          sync()
        end
        $ 4413 "Set CO[1]=Apagar"
        set_configurable_digital_out(1, False)
        $ 4414 "subir" "breakAfter"
        movel(subir, a=0.015, v=0.015)
        $ 4415 "bajada_broca≔pose_sub(bajada_broca, bajada)"
        global bajada_broca= pose_sub (bajada_broca, bajada)
        Loop_88 = Loop_88 + 1
      end
      $ 4416 "Direction: Base Z+"
      global move_thread_flag_4416=0
      thread move_thread_4416():
        enter_critical
        move_thread_flag_4416 = 1
        local towardsPos=calculate_point_to_move_towards(p[0.0,0.0,0.0,0.0,0.0,0.0], [0.0,0.0,1.0], 0.08)
        movel(towardsPos, a=0.15, v=0.1)
        move_thread_flag_4416 = 2
        exit_critical
      end
      move_thread_flag_4416 = 0
      move_thread_han_4416 = run move_thread_4416()
      while (True):
        sleep(1.0E-10)
        if (move_thread_flag_4416 > 1):
          join move_thread_han_4416
          $ 4417 "Until (distance)"
          break
        end
        sync()
      end
      $ 4418 "Set CO[1]=Apagar"
      set_configurable_digital_out(1, False)
      $ 4419 "barreno_actual≔barreno_actual+1"
      global barreno_actual=barreno_actual+1
    end
    $ 4422 "Popup: Linea23 con chica Terminada!"
    popup("Linea23 con chica Terminada!", "Mensaje", False, False, blocking=True)
    $ 4423 "Linea24"
    $ 4424 "Marcar_puntos"
    $ 4425 "MoveL"
    $ 4426 "Linea24_A" "breakAfter"
    movel(Linea24_A_p, a=0.5, v=0.1)
    $ 4427 "bajada_comprobacion"
    $ 4428 "Direction: Base Z-"
    global move_thread_flag_4428=0
    thread move_thread_4428():
      enter_critical
      move_thread_flag_4428 = 1
      local towardsPos=calculate_point_to_move_towards(p[0.0,0.0,0.0,0.0,0.0,0.0], [0.0,0.0,-1.0], 0.071)
      movel(towardsPos, a=0.15, v=0.1)
      move_thread_flag_4428 = 2
      exit_critical
    end
    move_thread_flag_4428 = 0
    move_thread_han_4428 = run move_thread_4428()
    while (True):
      sleep(1.0E-10)
      if (move_thread_flag_4428 > 1):
        join move_thread_han_4428
        $ 4429 "Until (distance)"
        break
      end
      sync()
    end
    $ 4430 "Direction: Base Z-"
    global move_thread_flag_4430=0
    thread move_thread_4430():
      enter_critical
      move_thread_flag_4430 = 1
      local towardsPos=calculate_point_to_move_towards(p[0.0,0.0,0.0,0.0,0.0,0.0], [0.0,0.0,-1.0], 1000.0)
      movel(towardsPos, a=0.007, v=0.007)
      move_thread_flag_4430 = 2
      exit_critical
    end
    move_thread_flag_4430 = 0
    move_thread_han_4430 = run move_thread_4430()
    while (True):
      local targetTcpDirection=get_target_tcp_speed()
      local stepsToRetract=tool_contact(direction=targetTcpDirection)
      if (stepsToRetract > 0):
        kill move_thread_han_4430
        stopl(0.02)
        local backTrackMovement=get_actual_joint_positions_history(stepsToRetract)
        local contactPose=get_forward_kin(backTrackMovement)
        local posDir=[targetTcpDirection[0],targetTcpDirection[1],targetTcpDirection[2]]
        local retractTo=contactPose
        if (norm(posDir) > 1e-6):
          local normalizedPosDir=normalize(posDir)
          local additionalRetraction=p[normalizedPosDir[0] * 0.0, normalizedPosDir[1] * 0.0, normalizedPosDir[2] * 0.0, 0, 0, 0]
          retractTo = pose_sub(contactPose, additionalRetraction)
        end
        movel(retractTo, a=0.02, v=0.1)
        $ 4431 "Until (tool_contact_detection)"
        break
      end
      sync()
    end
    $ 4432 "Direction: Base Z+"
    global move_thread_flag_4432=0
    thread move_thread_4432():
      enter_critical
      move_thread_flag_4432 = 1
      local towardsPos=calculate_point_to_move_towards(p[0.0,0.0,0.0,0.0,0.0,0.0], [0.0,0.0,1.0], 0.08)
      movel(towardsPos, a=0.15, v=0.1)
      move_thread_flag_4432 = 2
      exit_critical
    end
    move_thread_flag_4432 = 0
    move_thread_han_4432 = run move_thread_4432()
    while (True):
      sleep(1.0E-10)
      if (move_thread_flag_4432 > 1):
        join move_thread_han_4432
        $ 4433 "Until (distance)"
        break
      end
      sync()
    end
    $ 4434 "Linea24_B" "breakAfter"
    movel(Linea24_B_p, a=0.5, v=0.1)
    $ 4435 "bajada_comprobacion"
    $ 4436 "Direction: Base Z-"
    global move_thread_flag_4436=0
    thread move_thread_4436():
      enter_critical
      move_thread_flag_4436 = 1
      local towardsPos=calculate_point_to_move_towards(p[0.0,0.0,0.0,0.0,0.0,0.0], [0.0,0.0,-1.0], 0.071)
      movel(towardsPos, a=0.15, v=0.1)
      move_thread_flag_4436 = 2
      exit_critical
    end
    move_thread_flag_4436 = 0
    move_thread_han_4436 = run move_thread_4436()
    while (True):
      sleep(1.0E-10)
      if (move_thread_flag_4436 > 1):
        join move_thread_han_4436
        $ 4437 "Until (distance)"
        break
      end
      sync()
    end
    $ 4438 "Direction: Base Z-"
    global move_thread_flag_4438=0
    thread move_thread_4438():
      enter_critical
      move_thread_flag_4438 = 1
      local towardsPos=calculate_point_to_move_towards(p[0.0,0.0,0.0,0.0,0.0,0.0], [0.0,0.0,-1.0], 1000.0)
      movel(towardsPos, a=0.007, v=0.007)
      move_thread_flag_4438 = 2
      exit_critical
    end
    move_thread_flag_4438 = 0
    move_thread_han_4438 = run move_thread_4438()
    while (True):
      local targetTcpDirection=get_target_tcp_speed()
      local stepsToRetract=tool_contact(direction=targetTcpDirection)
      if (stepsToRetract > 0):
        kill move_thread_han_4438
        stopl(0.02)
        local backTrackMovement=get_actual_joint_positions_history(stepsToRetract)
        local contactPose=get_forward_kin(backTrackMovement)
        local posDir=[targetTcpDirection[0],targetTcpDirection[1],targetTcpDirection[2]]
        local retractTo=contactPose
        if (norm(posDir) > 1e-6):
          local normalizedPosDir=normalize(posDir)
          local additionalRetraction=p[normalizedPosDir[0] * 0.0, normalizedPosDir[1] * 0.0, normalizedPosDir[2] * 0.0, 0, 0, 0]
          retractTo = pose_sub(contactPose, additionalRetraction)
        end
        movel(retractTo, a=0.02, v=0.1)
        $ 4439 "Until (tool_contact_detection)"
        break
      end
      sync()
    end
    $ 4440 "Direction: Base Z+"
    global move_thread_flag_4440=0
    thread move_thread_4440():
      enter_critical
      move_thread_flag_4440 = 1
      local towardsPos=calculate_point_to_move_towards(p[0.0,0.0,0.0,0.0,0.0,0.0], [0.0,0.0,1.0], 0.08)
      movel(towardsPos, a=0.15, v=0.1)
      move_thread_flag_4440 = 2
      exit_critical
    end
    move_thread_flag_4440 = 0
    move_thread_han_4440 = run move_thread_4440()
    while (True):
      sleep(1.0E-10)
      if (move_thread_flag_4440 > 1):
        join move_thread_han_4440
        $ 4441 "Until (distance)"
        break
      end
      sync()
    end
    $ 4442 "AB"
    $ 4443 "'desbaste_inicial'"
    # 'desbaste_inicial'
    $ 4444 "bajada_broca≔p[0,0,-0.008,0,0,0]"
    global bajada_broca=p[0,0,-0.008,0,0,0]
    $ 4445 "barrenos_menos1≔4"
    global barrenos_menos1=4
    $ 4446 "barreno_actual≔0"
    global barreno_actual=0
    $ 4447 "Loop barreno_actual≤barrenos_menos1"
    while (barreno_actual <= barrenos_menos1):
      $ 4448 "Perforacion"
      $ 4449 "MoveL"
      $ 4450 "If barreno_actual≟2"
      if (barreno_actual == 2):
        $ 4451 "barreno_actual≔barreno_actual+1"
        global barreno_actual=barreno_actual+1
      end
      $ 4452 "internos≔interpolate_pose(Linea24_A, Linea24_B, barreno_actual/barrenos_menos1)"
      global internos= interpolate_pose (Linea24_A_p, Linea24_B_p, barreno_actual/barrenos_menos1)
      $ 4453 "internos" "breakAfter"
      movel(internos, a=0.5, v=0.1)
      $ 4454 "'desbaste_inicial'"
      # 'desbaste_inicial'
      $ 4455 "bajada_broca≔p[0,0,-0.024,0,0,0]"
      global bajada_broca=p[0,0,-0.024,0,0,0]
      $ 4456 "bajada≔p[0,0,0.024,0,0,0]"
      global bajada=p[0,0,0.024,0,0,0]
      $ 4457 "Direction: Base Z-"
      global move_thread_flag_4457=0
      thread move_thread_4457():
        enter_critical
        move_thread_flag_4457 = 1
        local towardsPos=calculate_point_to_move_towards(p[0.0,0.0,0.0,0.0,0.0,0.0], [0.0,0.0,-1.0], 0.071)
        movel(towardsPos, a=0.15, v=0.1)
        move_thread_flag_4457 = 2
        exit_critical
      end
      move_thread_flag_4457 = 0
      move_thread_han_4457 = run move_thread_4457()
      while (True):
        sleep(1.0E-10)
        if (move_thread_flag_4457 > 1):
          join move_thread_han_4457
          $ 4458 "Until (distance)"
          break
        end
        sync()
      end
      $ 4459 "Direction: Base Z-"
      global move_thread_flag_4459=0
      thread move_thread_4459():
        enter_critical
        move_thread_flag_4459 = 1
        local towardsPos=calculate_point_to_move_towards(p[0.0,0.0,0.0,0.0,0.0,0.0], [0.0,0.0,-1.0], 1000.0)
        movel(towardsPos, a=0.007, v=0.007)
        move_thread_flag_4459 = 2
        exit_critical
      end
      move_thread_flag_4459 = 0
      move_thread_han_4459 = run move_thread_4459()
      while (True):
        local targetTcpDirection=get_target_tcp_speed()
        local stepsToRetract=tool_contact(direction=targetTcpDirection)
        if (stepsToRetract > 0):
          kill move_thread_han_4459
          stopl(0.02)
          local backTrackMovement=get_actual_joint_positions_history(stepsToRetract)
          local contactPose=get_forward_kin(backTrackMovement)
          local posDir=[targetTcpDirection[0],targetTcpDirection[1],targetTcpDirection[2]]
          local retractTo=contactPose
          if (norm(posDir) > 1e-6):
            local normalizedPosDir=normalize(posDir)
            local additionalRetraction=p[normalizedPosDir[0] * 0.0, normalizedPosDir[1] * 0.0, normalizedPosDir[2] * 0.0, 0, 0, 0]
            retractTo = pose_sub(contactPose, additionalRetraction)
          end
          movel(retractTo, a=0.02, v=0.1)
          $ 4460 "Until (tool_contact_detection)"
          break
        end
        sync()
      end
      $ 4461 "Popup: punto contacto alanzdo"
      popup("punto contacto alanzdo", "Mensaje", False, False, blocking=True)
      $ 4462 "Direction: Base Z+"
      global move_thread_flag_4462=0
      thread move_thread_4462():
        enter_critical
        move_thread_flag_4462 = 1
        local towardsPos=calculate_point_to_move_towards(p[0.0,0.0,0.0,0.0,0.0,0.0], [0.0,0.0,1.0], 0.007)
        movel(towardsPos, a=0.015, v=0.015)
        move_thread_flag_4462 = 2
        exit_critical
      end
      move_thread_flag_4462 = 0
      move_thread_han_4462 = run move_thread_4462()
      while (True):
        sleep(1.0E-10)
        if (move_thread_flag_4462 > 1):
          join move_thread_han_4462
          $ 4463 "Until (distance)"
          break
        end
        sync()
      end
      $ 4464 "Wait: 0.3"
      sleep(0.3)
      $ 4465 "Set CO[1]=Encender"
      set_configurable_digital_out(1, True)
      $ 4466 "Wait: 0.3"
      sleep(0.3)
      $ 4467 "Loop 1 times"
      Loop_102 = 0
      while (Loop_102 < 1):
        $ 4468 "bajar≔pose_add(get_actual_tcp_pose(), bajada_broca)"
        global bajar= pose_add ( get_actual_tcp_pose (), bajada_broca)
        $ 4469 "bajar" "breakAfter"
        movel(bajar, a=0.004, v=0.004)
        $ 4470 "subir≔pose_sub(get_actual_tcp_pose(), bajada_broca)"
        global subir= pose_sub ( get_actual_tcp_pose (), bajada_broca)
        $ 4471 "Direction: Base Z+"
        global move_thread_flag_4471=0
        thread move_thread_4471():
          enter_critical
          move_thread_flag_4471 = 1
          local towardsPos=calculate_point_to_move_towards(p[0.0,0.0,0.0,0.0,0.0,0.0], [0.0,0.0,1.0], 0.002)
          movel(towardsPos, a=0.015, v=0.015)
          move_thread_flag_4471 = 2
          exit_critical
        end
        move_thread_flag_4471 = 0
        move_thread_han_4471 = run move_thread_4471()
        while (True):
          sleep(1.0E-10)
          if (move_thread_flag_4471 > 1):
            join move_thread_han_4471
            $ 4472 "Until (distance)"
            break
          end
          sync()
        end
        $ 4473 "Set CO[1]=Apagar"
        set_configurable_digital_out(1, False)
        $ 4474 "subir" "breakAfter"
        movel(subir, a=0.015, v=0.015)
        $ 4475 "bajada_broca≔pose_sub(bajada_broca, bajada)"
        global bajada_broca= pose_sub (bajada_broca, bajada)
        Loop_102 = Loop_102 + 1
      end
      $ 4476 "Direction: Base Z+"
      global move_thread_flag_4476=0
      thread move_thread_4476():
        enter_critical
        move_thread_flag_4476 = 1
        local towardsPos=calculate_point_to_move_towards(p[0.0,0.0,0.0,0.0,0.0,0.0], [0.0,0.0,1.0], 0.08)
        movel(towardsPos, a=0.15, v=0.1)
        move_thread_flag_4476 = 2
        exit_critical
      end
      move_thread_flag_4476 = 0
      move_thread_han_4476 = run move_thread_4476()
      while (True):
        sleep(1.0E-10)
        if (move_thread_flag_4476 > 1):
          join move_thread_han_4476
          $ 4477 "Until (distance)"
          break
        end
        sync()
      end
      $ 4478 "Set CO[1]=Apagar"
      set_configurable_digital_out(1, False)
      $ 4479 "barreno_actual≔barreno_actual+1"
      global barreno_actual=barreno_actual+1
    end
    $ 4482 "Popup: Linea24 con chica Terminada!"
    popup("Linea24 con chica Terminada!", "Mensaje", False, False, blocking=True)
    $ 4483 "Linea25"
    $ 4484 "Marcar_puntos"
    $ 4485 "MoveL"
    $ 4486 "Linea25_A" "breakAfter"
    movel(Linea25_A_p, a=0.5, v=0.1)
    $ 4487 "bajada_comprobacion"
    $ 4488 "Direction: Base Z-"
    global move_thread_flag_4488=0
    thread move_thread_4488():
      enter_critical
      move_thread_flag_4488 = 1
      local towardsPos=calculate_point_to_move_towards(p[0.0,0.0,0.0,0.0,0.0,0.0], [0.0,0.0,-1.0], 0.071)
      movel(towardsPos, a=0.15, v=0.1)
      move_thread_flag_4488 = 2
      exit_critical
    end
    move_thread_flag_4488 = 0
    move_thread_han_4488 = run move_thread_4488()
    while (True):
      sleep(1.0E-10)
      if (move_thread_flag_4488 > 1):
        join move_thread_han_4488
        $ 4489 "Until (distance)"
        break
      end
      sync()
    end
    $ 4490 "Direction: Base Z-"
    global move_thread_flag_4490=0
    thread move_thread_4490():
      enter_critical
      move_thread_flag_4490 = 1
      local towardsPos=calculate_point_to_move_towards(p[0.0,0.0,0.0,0.0,0.0,0.0], [0.0,0.0,-1.0], 1000.0)
      movel(towardsPos, a=0.007, v=0.007)
      move_thread_flag_4490 = 2
      exit_critical
    end
    move_thread_flag_4490 = 0
    move_thread_han_4490 = run move_thread_4490()
    while (True):
      local targetTcpDirection=get_target_tcp_speed()
      local stepsToRetract=tool_contact(direction=targetTcpDirection)
      if (stepsToRetract > 0):
        kill move_thread_han_4490
        stopl(0.02)
        local backTrackMovement=get_actual_joint_positions_history(stepsToRetract)
        local contactPose=get_forward_kin(backTrackMovement)
        local posDir=[targetTcpDirection[0],targetTcpDirection[1],targetTcpDirection[2]]
        local retractTo=contactPose
        if (norm(posDir) > 1e-6):
          local normalizedPosDir=normalize(posDir)
          local additionalRetraction=p[normalizedPosDir[0] * 0.0, normalizedPosDir[1] * 0.0, normalizedPosDir[2] * 0.0, 0, 0, 0]
          retractTo = pose_sub(contactPose, additionalRetraction)
        end
        movel(retractTo, a=0.02, v=0.1)
        $ 4491 "Until (tool_contact_detection)"
        break
      end
      sync()
    end
    $ 4492 "Direction: Base Z+"
    global move_thread_flag_4492=0
    thread move_thread_4492():
      enter_critical
      move_thread_flag_4492 = 1
      local towardsPos=calculate_point_to_move_towards(p[0.0,0.0,0.0,0.0,0.0,0.0], [0.0,0.0,1.0], 0.08)
      movel(towardsPos, a=0.15, v=0.1)
      move_thread_flag_4492 = 2
      exit_critical
    end
    move_thread_flag_4492 = 0
    move_thread_han_4492 = run move_thread_4492()
    while (True):
      sleep(1.0E-10)
      if (move_thread_flag_4492 > 1):
        join move_thread_han_4492
        $ 4493 "Until (distance)"
        break
      end
      sync()
    end
    $ 4494 "Linea25_B" "breakAfter"
    movel(Linea25_B_p, a=0.5, v=0.1)
    $ 4495 "bajada_comprobacion"
    $ 4496 "Direction: Base Z-"
    global move_thread_flag_4496=0
    thread move_thread_4496():
      enter_critical
      move_thread_flag_4496 = 1
      local towardsPos=calculate_point_to_move_towards(p[0.0,0.0,0.0,0.0,0.0,0.0], [0.0,0.0,-1.0], 0.071)
      movel(towardsPos, a=0.15, v=0.1)
      move_thread_flag_4496 = 2
      exit_critical
    end
    move_thread_flag_4496 = 0
    move_thread_han_4496 = run move_thread_4496()
    while (True):
      sleep(1.0E-10)
      if (move_thread_flag_4496 > 1):
        join move_thread_han_4496
        $ 4497 "Until (distance)"
        break
      end
      sync()
    end
    $ 4498 "Direction: Base Z-"
    global move_thread_flag_4498=0
    thread move_thread_4498():
      enter_critical
      move_thread_flag_4498 = 1
      local towardsPos=calculate_point_to_move_towards(p[0.0,0.0,0.0,0.0,0.0,0.0], [0.0,0.0,-1.0], 1000.0)
      movel(towardsPos, a=0.007, v=0.007)
      move_thread_flag_4498 = 2
      exit_critical
    end
    move_thread_flag_4498 = 0
    move_thread_han_4498 = run move_thread_4498()
    while (True):
      local targetTcpDirection=get_target_tcp_speed()
      local stepsToRetract=tool_contact(direction=targetTcpDirection)
      if (stepsToRetract > 0):
        kill move_thread_han_4498
        stopl(0.02)
        local backTrackMovement=get_actual_joint_positions_history(stepsToRetract)
        local contactPose=get_forward_kin(backTrackMovement)
        local posDir=[targetTcpDirection[0],targetTcpDirection[1],targetTcpDirection[2]]
        local retractTo=contactPose
        if (norm(posDir) > 1e-6):
          local normalizedPosDir=normalize(posDir)
          local additionalRetraction=p[normalizedPosDir[0] * 0.0, normalizedPosDir[1] * 0.0, normalizedPosDir[2] * 0.0, 0, 0, 0]
          retractTo = pose_sub(contactPose, additionalRetraction)
        end
        movel(retractTo, a=0.02, v=0.1)
        $ 4499 "Until (tool_contact_detection)"
        break
      end
      sync()
    end
    $ 4500 "Direction: Base Z+"
    global move_thread_flag_4500=0
    thread move_thread_4500():
      enter_critical
      move_thread_flag_4500 = 1
      local towardsPos=calculate_point_to_move_towards(p[0.0,0.0,0.0,0.0,0.0,0.0], [0.0,0.0,1.0], 0.08)
      movel(towardsPos, a=0.15, v=0.1)
      move_thread_flag_4500 = 2
      exit_critical
    end
    move_thread_flag_4500 = 0
    move_thread_han_4500 = run move_thread_4500()
    while (True):
      sleep(1.0E-10)
      if (move_thread_flag_4500 > 1):
        join move_thread_han_4500
        $ 4501 "Until (distance)"
        break
      end
      sync()
    end
    $ 4502 "AB"
    $ 4503 "'desbaste_inicial'"
    # 'desbaste_inicial'
    $ 4504 "bajada_broca≔p[0,0,-0.008,0,0,0]"
    global bajada_broca=p[0,0,-0.008,0,0,0]
    $ 4505 "barrenos_menos1≔2"
    global barrenos_menos1=2
    $ 4506 "barreno_actual≔0"
    global barreno_actual=0
    $ 4507 "Loop barreno_actual≤barrenos_menos1"
    while (barreno_actual <= barrenos_menos1):
      $ 4508 "Perforacion"
      $ 4509 "MoveL"
      $ 4512 "internos≔interpolate_pose(Linea25_A, Linea25_B, barreno_actual/barrenos_menos1)"
      global internos= interpolate_pose (Linea25_A_p, Linea25_B_p, barreno_actual/barrenos_menos1)
      $ 4513 "internos" "breakAfter"
      movel(internos, a=0.5, v=0.1)
      $ 4514 "'desbaste_inicial'"
      # 'desbaste_inicial'
      $ 4515 "bajada_broca≔p[0,0,-0.024,0,0,0]"
      global bajada_broca=p[0,0,-0.024,0,0,0]
      $ 4516 "bajada≔p[0,0,0.024,0,0,0]"
      global bajada=p[0,0,0.024,0,0,0]
      $ 4517 "Direction: Base Z-"
      global move_thread_flag_4517=0
      thread move_thread_4517():
        enter_critical
        move_thread_flag_4517 = 1
        local towardsPos=calculate_point_to_move_towards(p[0.0,0.0,0.0,0.0,0.0,0.0], [0.0,0.0,-1.0], 0.071)
        movel(towardsPos, a=0.15, v=0.1)
        move_thread_flag_4517 = 2
        exit_critical
      end
      move_thread_flag_4517 = 0
      move_thread_han_4517 = run move_thread_4517()
      while (True):
        sleep(1.0E-10)
        if (move_thread_flag_4517 > 1):
          join move_thread_han_4517
          $ 4518 "Until (distance)"
          break
        end
        sync()
      end
      $ 4519 "Direction: Base Z-"
      global move_thread_flag_4519=0
      thread move_thread_4519():
        enter_critical
        move_thread_flag_4519 = 1
        local towardsPos=calculate_point_to_move_towards(p[0.0,0.0,0.0,0.0,0.0,0.0], [0.0,0.0,-1.0], 1000.0)
        movel(towardsPos, a=0.007, v=0.007)
        move_thread_flag_4519 = 2
        exit_critical
      end
      move_thread_flag_4519 = 0
      move_thread_han_4519 = run move_thread_4519()
      while (True):
        local targetTcpDirection=get_target_tcp_speed()
        local stepsToRetract=tool_contact(direction=targetTcpDirection)
        if (stepsToRetract > 0):
          kill move_thread_han_4519
          stopl(0.02)
          local backTrackMovement=get_actual_joint_positions_history(stepsToRetract)
          local contactPose=get_forward_kin(backTrackMovement)
          local posDir=[targetTcpDirection[0],targetTcpDirection[1],targetTcpDirection[2]]
          local retractTo=contactPose
          if (norm(posDir) > 1e-6):
            local normalizedPosDir=normalize(posDir)
            local additionalRetraction=p[normalizedPosDir[0] * 0.0, normalizedPosDir[1] * 0.0, normalizedPosDir[2] * 0.0, 0, 0, 0]
            retractTo = pose_sub(contactPose, additionalRetraction)
          end
          movel(retractTo, a=0.02, v=0.1)
          $ 4520 "Until (tool_contact_detection)"
          break
        end
        sync()
      end
      $ 4521 "Popup: punto contacto alanzdo"
      popup("punto contacto alanzdo", "Mensaje", False, False, blocking=True)
      $ 4522 "Direction: Base Z+"
      global move_thread_flag_4522=0
      thread move_thread_4522():
        enter_critical
        move_thread_flag_4522 = 1
        local towardsPos=calculate_point_to_move_towards(p[0.0,0.0,0.0,0.0,0.0,0.0], [0.0,0.0,1.0], 0.007)
        movel(towardsPos, a=0.015, v=0.015)
        move_thread_flag_4522 = 2
        exit_critical
      end
      move_thread_flag_4522 = 0
      move_thread_han_4522 = run move_thread_4522()
      while (True):
        sleep(1.0E-10)
        if (move_thread_flag_4522 > 1):
          join move_thread_han_4522
          $ 4523 "Until (distance)"
          break
        end
        sync()
      end
      $ 4524 "Wait: 0.3"
      sleep(0.3)
      $ 4525 "Set CO[1]=Encender"
      set_configurable_digital_out(1, True)
      $ 4526 "Wait: 0.3"
      sleep(0.3)
      $ 4527 "Loop 1 times"
      Loop_135 = 0
      while (Loop_135 < 1):
        $ 4528 "bajar≔pose_add(get_actual_tcp_pose(), bajada_broca)"
        global bajar= pose_add ( get_actual_tcp_pose (), bajada_broca)
        $ 4529 "bajar" "breakAfter"
        movel(bajar, a=0.004, v=0.004)
        $ 4530 "subir≔pose_sub(get_actual_tcp_pose(), bajada_broca)"
        global subir= pose_sub ( get_actual_tcp_pose (), bajada_broca)
        $ 4531 "Direction: Base Z+"
        global move_thread_flag_4531=0
        thread move_thread_4531():
          enter_critical
          move_thread_flag_4531 = 1
          local towardsPos=calculate_point_to_move_towards(p[0.0,0.0,0.0,0.0,0.0,0.0], [0.0,0.0,1.0], 0.002)
          movel(towardsPos, a=0.015, v=0.015)
          move_thread_flag_4531 = 2
          exit_critical
        end
        move_thread_flag_4531 = 0
        move_thread_han_4531 = run move_thread_4531()
        while (True):
          sleep(1.0E-10)
          if (move_thread_flag_4531 > 1):
            join move_thread_han_4531
            $ 4532 "Until (distance)"
            break
          end
          sync()
        end
        $ 4533 "Set CO[1]=Apagar"
        set_configurable_digital_out(1, False)
        $ 4534 "subir" "breakAfter"
        movel(subir, a=0.015, v=0.015)
        $ 4535 "bajada_broca≔pose_sub(bajada_broca, bajada)"
        global bajada_broca= pose_sub (bajada_broca, bajada)
        Loop_135 = Loop_135 + 1
      end
      $ 4536 "Direction: Base Z+"
      global move_thread_flag_4536=0
      thread move_thread_4536():
        enter_critical
        move_thread_flag_4536 = 1
        local towardsPos=calculate_point_to_move_towards(p[0.0,0.0,0.0,0.0,0.0,0.0], [0.0,0.0,1.0], 0.08)
        movel(towardsPos, a=0.15, v=0.1)
        move_thread_flag_4536 = 2
        exit_critical
      end
      move_thread_flag_4536 = 0
      move_thread_han_4536 = run move_thread_4536()
      while (True):
        sleep(1.0E-10)
        if (move_thread_flag_4536 > 1):
          join move_thread_han_4536
          $ 4537 "Until (distance)"
          break
        end
        sync()
      end
      $ 4538 "Set CO[1]=Apagar"
      set_configurable_digital_out(1, False)
      $ 4539 "barreno_actual≔barreno_actual+1"
      global barreno_actual=barreno_actual+1
    end
    $ 4542 "Popup: Linea25 con chica Terminada!"
    popup("Linea25 con chica Terminada!", "Mensaje", False, False, blocking=True)
    $ 4543 "Linea26"
    $ 4544 "Marcar_puntos"
    $ 4545 "MoveL"
    $ 4546 "Linea26_A" "breakAfter"
    movel(Linea26_A_p, a=0.5, v=0.1)
    $ 4547 "bajada_comprobacion"
    $ 4548 "Direction: Base Z-"
    global move_thread_flag_4548=0
    thread move_thread_4548():
      enter_critical
      move_thread_flag_4548 = 1
      local towardsPos=calculate_point_to_move_towards(p[0.0,0.0,0.0,0.0,0.0,0.0], [0.0,0.0,-1.0], 0.071)
      movel(towardsPos, a=0.15, v=0.1)
      move_thread_flag_4548 = 2
      exit_critical
    end
    move_thread_flag_4548 = 0
    move_thread_han_4548 = run move_thread_4548()
    while (True):
      sleep(1.0E-10)
      if (move_thread_flag_4548 > 1):
        join move_thread_han_4548
        $ 4549 "Until (distance)"
        break
      end
      sync()
    end
    $ 4550 "Direction: Base Z-"
    global move_thread_flag_4550=0
    thread move_thread_4550():
      enter_critical
      move_thread_flag_4550 = 1
      local towardsPos=calculate_point_to_move_towards(p[0.0,0.0,0.0,0.0,0.0,0.0], [0.0,0.0,-1.0], 1000.0)
      movel(towardsPos, a=0.007, v=0.007)
      move_thread_flag_4550 = 2
      exit_critical
    end
    move_thread_flag_4550 = 0
    move_thread_han_4550 = run move_thread_4550()
    while (True):
      local targetTcpDirection=get_target_tcp_speed()
      local stepsToRetract=tool_contact(direction=targetTcpDirection)
      if (stepsToRetract > 0):
        kill move_thread_han_4550
        stopl(0.02)
        local backTrackMovement=get_actual_joint_positions_history(stepsToRetract)
        local contactPose=get_forward_kin(backTrackMovement)
        local posDir=[targetTcpDirection[0],targetTcpDirection[1],targetTcpDirection[2]]
        local retractTo=contactPose
        if (norm(posDir) > 1e-6):
          local normalizedPosDir=normalize(posDir)
          local additionalRetraction=p[normalizedPosDir[0] * 0.0, normalizedPosDir[1] * 0.0, normalizedPosDir[2] * 0.0, 0, 0, 0]
          retractTo = pose_sub(contactPose, additionalRetraction)
        end
        movel(retractTo, a=0.02, v=0.1)
        $ 4551 "Until (tool_contact_detection)"
        break
      end
      sync()
    end
    $ 4552 "Direction: Base Z+"
    global move_thread_flag_4552=0
    thread move_thread_4552():
      enter_critical
      move_thread_flag_4552 = 1
      local towardsPos=calculate_point_to_move_towards(p[0.0,0.0,0.0,0.0,0.0,0.0], [0.0,0.0,1.0], 0.08)
      movel(towardsPos, a=0.15, v=0.1)
      move_thread_flag_4552 = 2
      exit_critical
    end
    move_thread_flag_4552 = 0
    move_thread_han_4552 = run move_thread_4552()
    while (True):
      sleep(1.0E-10)
      if (move_thread_flag_4552 > 1):
        join move_thread_han_4552
        $ 4553 "Until (distance)"
        break
      end
      sync()
    end
    $ 4554 "Linea26_B" "breakAfter"
    movel(Linea26_B_p, a=0.5, v=0.1)
    $ 4555 "bajada_comprobacion"
    $ 4556 "Direction: Base Z-"
    global move_thread_flag_4556=0
    thread move_thread_4556():
      enter_critical
      move_thread_flag_4556 = 1
      local towardsPos=calculate_point_to_move_towards(p[0.0,0.0,0.0,0.0,0.0,0.0], [0.0,0.0,-1.0], 0.071)
      movel(towardsPos, a=0.15, v=0.1)
      move_thread_flag_4556 = 2
      exit_critical
    end
    move_thread_flag_4556 = 0
    move_thread_han_4556 = run move_thread_4556()
    while (True):
      sleep(1.0E-10)
      if (move_thread_flag_4556 > 1):
        join move_thread_han_4556
        $ 4557 "Until (distance)"
        break
      end
      sync()
    end
    $ 4558 "Direction: Base Z-"
    global move_thread_flag_4558=0
    thread move_thread_4558():
      enter_critical
      move_thread_flag_4558 = 1
      local towardsPos=calculate_point_to_move_towards(p[0.0,0.0,0.0,0.0,0.0,0.0], [0.0,0.0,-1.0], 1000.0)
      movel(towardsPos, a=0.007, v=0.007)
      move_thread_flag_4558 = 2
      exit_critical
    end
    move_thread_flag_4558 = 0
    move_thread_han_4558 = run move_thread_4558()
    while (True):
      local targetTcpDirection=get_target_tcp_speed()
      local stepsToRetract=tool_contact(direction=targetTcpDirection)
      if (stepsToRetract > 0):
        kill move_thread_han_4558
        stopl(0.02)
        local backTrackMovement=get_actual_joint_positions_history(stepsToRetract)
        local contactPose=get_forward_kin(backTrackMovement)
        local posDir=[targetTcpDirection[0],targetTcpDirection[1],targetTcpDirection[2]]
        local retractTo=contactPose
        if (norm(posDir) > 1e-6):
          local normalizedPosDir=normalize(posDir)
          local additionalRetraction=p[normalizedPosDir[0] * 0.0, normalizedPosDir[1] * 0.0, normalizedPosDir[2] * 0.0, 0, 0, 0]
          retractTo = pose_sub(contactPose, additionalRetraction)
        end
        movel(retractTo, a=0.02, v=0.1)
        $ 4559 "Until (tool_contact_detection)"
        break
      end
      sync()
    end
    $ 4560 "Direction: Base Z+"
    global move_thread_flag_4560=0
    thread move_thread_4560():
      enter_critical
      move_thread_flag_4560 = 1
      local towardsPos=calculate_point_to_move_towards(p[0.0,0.0,0.0,0.0,0.0,0.0], [0.0,0.0,1.0], 0.08)
      movel(towardsPos, a=0.15, v=0.1)
      move_thread_flag_4560 = 2
      exit_critical
    end
    move_thread_flag_4560 = 0
    move_thread_han_4560 = run move_thread_4560()
    while (True):
      sleep(1.0E-10)
      if (move_thread_flag_4560 > 1):
        join move_thread_han_4560
        $ 4561 "Until (distance)"
        break
      end
      sync()
    end
    $ 4562 "AB"
    $ 4563 "'desbaste_inicial'"
    # 'desbaste_inicial'
    $ 4564 "bajada_broca≔p[0,0,-0.008,0,0,0]"
    global bajada_broca=p[0,0,-0.008,0,0,0]
    $ 4565 "barrenos_menos1≔1"
    global barrenos_menos1=1
    $ 4566 "barreno_actual≔0"
    global barreno_actual=0
    $ 4567 "Loop barreno_actual≤barrenos_menos1"
    while (barreno_actual <= barrenos_menos1):
      $ 4568 "Perforacion"
      $ 4569 "MoveL"
      $ 4572 "internos≔interpolate_pose(Linea26_A, Linea26_B, barreno_actual/barrenos_menos1)"
      global internos= interpolate_pose (Linea26_A_p, Linea26_B_p, barreno_actual/barrenos_menos1)
      $ 4573 "internos" "breakAfter"
      movel(internos, a=0.5, v=0.1)
      $ 4574 "'desbaste_inicial'"
      # 'desbaste_inicial'
      $ 4575 "bajada_broca≔p[0,0,-0.024,0,0,0]"
      global bajada_broca=p[0,0,-0.024,0,0,0]
      $ 4576 "bajada≔p[0,0,0.024,0,0,0]"
      global bajada=p[0,0,0.024,0,0,0]
      $ 4577 "Direction: Base Z-"
      global move_thread_flag_4577=0
      thread move_thread_4577():
        enter_critical
        move_thread_flag_4577 = 1
        local towardsPos=calculate_point_to_move_towards(p[0.0,0.0,0.0,0.0,0.0,0.0], [0.0,0.0,-1.0], 0.071)
        movel(towardsPos, a=0.15, v=0.1)
        move_thread_flag_4577 = 2
        exit_critical
      end
      move_thread_flag_4577 = 0
      move_thread_han_4577 = run move_thread_4577()
      while (True):
        sleep(1.0E-10)
        if (move_thread_flag_4577 > 1):
          join move_thread_han_4577
          $ 4578 "Until (distance)"
          break
        end
        sync()
      end
      $ 4579 "Direction: Base Z-"
      global move_thread_flag_4579=0
      thread move_thread_4579():
        enter_critical
        move_thread_flag_4579 = 1
        local towardsPos=calculate_point_to_move_towards(p[0.0,0.0,0.0,0.0,0.0,0.0], [0.0,0.0,-1.0], 1000.0)
        movel(towardsPos, a=0.007, v=0.007)
        move_thread_flag_4579 = 2
        exit_critical
      end
      move_thread_flag_4579 = 0
      move_thread_han_4579 = run move_thread_4579()
      while (True):
        local targetTcpDirection=get_target_tcp_speed()
        local stepsToRetract=tool_contact(direction=targetTcpDirection)
        if (stepsToRetract > 0):
          kill move_thread_han_4579
          stopl(0.02)
          local backTrackMovement=get_actual_joint_positions_history(stepsToRetract)
          local contactPose=get_forward_kin(backTrackMovement)
          local posDir=[targetTcpDirection[0],targetTcpDirection[1],targetTcpDirection[2]]
          local retractTo=contactPose
          if (norm(posDir) > 1e-6):
            local normalizedPosDir=normalize(posDir)
            local additionalRetraction=p[normalizedPosDir[0] * 0.0, normalizedPosDir[1] * 0.0, normalizedPosDir[2] * 0.0, 0, 0, 0]
            retractTo = pose_sub(contactPose, additionalRetraction)
          end
          movel(retractTo, a=0.02, v=0.1)
          $ 4580 "Until (tool_contact_detection)"
          break
        end
        sync()
      end
      $ 4581 "Popup: punto contacto alanzdo"
      popup("punto contacto alanzdo", "Mensaje", False, False, blocking=True)
      $ 4582 "Direction: Base Z+"
      global move_thread_flag_4582=0
      thread move_thread_4582():
        enter_critical
        move_thread_flag_4582 = 1
        local towardsPos=calculate_point_to_move_towards(p[0.0,0.0,0.0,0.0,0.0,0.0], [0.0,0.0,1.0], 0.007)
        movel(towardsPos, a=0.015, v=0.015)
        move_thread_flag_4582 = 2
        exit_critical
      end
      move_thread_flag_4582 = 0
      move_thread_han_4582 = run move_thread_4582()
      while (True):
        sleep(1.0E-10)
        if (move_thread_flag_4582 > 1):
          join move_thread_han_4582
          $ 4583 "Until (distance)"
          break
        end
        sync()
      end
      $ 4584 "Wait: 0.3"
      sleep(0.3)
      $ 4585 "Set CO[1]=Encender"
      set_configurable_digital_out(1, True)
      $ 4586 "Wait: 0.3"
      sleep(0.3)
      $ 4587 "Loop 1 times"
      Loop_138 = 0
      while (Loop_138 < 1):
        $ 4588 "bajar≔pose_add(get_actual_tcp_pose(), bajada_broca)"
        global bajar= pose_add ( get_actual_tcp_pose (), bajada_broca)
        $ 4589 "bajar" "breakAfter"
        movel(bajar, a=0.004, v=0.004)
        $ 4590 "subir≔pose_sub(get_actual_tcp_pose(), bajada_broca)"
        global subir= pose_sub ( get_actual_tcp_pose (), bajada_broca)
        $ 4591 "Direction: Base Z+"
        global move_thread_flag_4591=0
        thread move_thread_4591():
          enter_critical
          move_thread_flag_4591 = 1
          local towardsPos=calculate_point_to_move_towards(p[0.0,0.0,0.0,0.0,0.0,0.0], [0.0,0.0,1.0], 0.002)
          movel(towardsPos, a=0.015, v=0.015)
          move_thread_flag_4591 = 2
          exit_critical
        end
        move_thread_flag_4591 = 0
        move_thread_han_4591 = run move_thread_4591()
        while (True):
          sleep(1.0E-10)
          if (move_thread_flag_4591 > 1):
            join move_thread_han_4591
            $ 4592 "Until (distance)"
            break
          end
          sync()
        end
        $ 4593 "Set CO[1]=Apagar"
        set_configurable_digital_out(1, False)
        $ 4594 "subir" "breakAfter"
        movel(subir, a=0.015, v=0.015)
        $ 4595 "bajada_broca≔pose_sub(bajada_broca, bajada)"
        global bajada_broca= pose_sub (bajada_broca, bajada)
        Loop_138 = Loop_138 + 1
      end
      $ 4596 "Direction: Base Z+"
      global move_thread_flag_4596=0
      thread move_thread_4596():
        enter_critical
        move_thread_flag_4596 = 1
        local towardsPos=calculate_point_to_move_towards(p[0.0,0.0,0.0,0.0,0.0,0.0], [0.0,0.0,1.0], 0.08)
        movel(towardsPos, a=0.15, v=0.1)
        move_thread_flag_4596 = 2
        exit_critical
      end
      move_thread_flag_4596 = 0
      move_thread_han_4596 = run move_thread_4596()
      while (True):
        sleep(1.0E-10)
        if (move_thread_flag_4596 > 1):
          join move_thread_han_4596
          $ 4597 "Until (distance)"
          break
        end
        sync()
      end
      $ 4598 "Set CO[1]=Apagar"
      set_configurable_digital_out(1, False)
      $ 4599 "barreno_actual≔barreno_actual+1"
      global barreno_actual=barreno_actual+1
    end
    $ 4602 "Popup: Linea26 con chica Terminada!"
    popup("Linea26 con chica Terminada!", "Mensaje", False, False, blocking=True)
    $ 4603 "Linea27"
    $ 4604 "Marcar_puntos"
    $ 4605 "MoveL"
    $ 4606 "Linea27_A" "breakAfter"
    movel(Linea27_A_p, a=0.5, v=0.1)
    $ 4607 "bajada_comprobacion"
    $ 4608 "Direction: Base Z-"
    global move_thread_flag_4608=0
    thread move_thread_4608():
      enter_critical
      move_thread_flag_4608 = 1
      local towardsPos=calculate_point_to_move_towards(p[0.0,0.0,0.0,0.0,0.0,0.0], [0.0,0.0,-1.0], 0.071)
      movel(towardsPos, a=0.15, v=0.1)
      move_thread_flag_4608 = 2
      exit_critical
    end
    move_thread_flag_4608 = 0
    move_thread_han_4608 = run move_thread_4608()
    while (True):
      sleep(1.0E-10)
      if (move_thread_flag_4608 > 1):
        join move_thread_han_4608
        $ 4609 "Until (distance)"
        break
      end
      sync()
    end
    $ 4610 "Direction: Base Z-"
    global move_thread_flag_4610=0
    thread move_thread_4610():
      enter_critical
      move_thread_flag_4610 = 1
      local towardsPos=calculate_point_to_move_towards(p[0.0,0.0,0.0,0.0,0.0,0.0], [0.0,0.0,-1.0], 1000.0)
      movel(towardsPos, a=0.007, v=0.007)
      move_thread_flag_4610 = 2
      exit_critical
    end
    move_thread_flag_4610 = 0
    move_thread_han_4610 = run move_thread_4610()
    while (True):
      local targetTcpDirection=get_target_tcp_speed()
      local stepsToRetract=tool_contact(direction=targetTcpDirection)
      if (stepsToRetract > 0):
        kill move_thread_han_4610
        stopl(0.02)
        local backTrackMovement=get_actual_joint_positions_history(stepsToRetract)
        local contactPose=get_forward_kin(backTrackMovement)
        local posDir=[targetTcpDirection[0],targetTcpDirection[1],targetTcpDirection[2]]
        local retractTo=contactPose
        if (norm(posDir) > 1e-6):
          local normalizedPosDir=normalize(posDir)
          local additionalRetraction=p[normalizedPosDir[0] * 0.0, normalizedPosDir[1] * 0.0, normalizedPosDir[2] * 0.0, 0, 0, 0]
          retractTo = pose_sub(contactPose, additionalRetraction)
        end
        movel(retractTo, a=0.02, v=0.1)
        $ 4611 "Until (tool_contact_detection)"
        break
      end
      sync()
    end
    $ 4612 "Direction: Base Z+"
    global move_thread_flag_4612=0
    thread move_thread_4612():
      enter_critical
      move_thread_flag_4612 = 1
      local towardsPos=calculate_point_to_move_towards(p[0.0,0.0,0.0,0.0,0.0,0.0], [0.0,0.0,1.0], 0.08)
      movel(towardsPos, a=0.15, v=0.1)
      move_thread_flag_4612 = 2
      exit_critical
    end
    move_thread_flag_4612 = 0
    move_thread_han_4612 = run move_thread_4612()
    while (True):
      sleep(1.0E-10)
      if (move_thread_flag_4612 > 1):
        join move_thread_han_4612
        $ 4613 "Until (distance)"
        break
      end
      sync()
    end
    $ 4614 "Linea27_B" "breakAfter"
    movel(Linea27_B_p, a=0.5, v=0.1)
    $ 4615 "bajada_comprobacion"
    $ 4616 "Direction: Base Z-"
    global move_thread_flag_4616=0
    thread move_thread_4616():
      enter_critical
      move_thread_flag_4616 = 1
      local towardsPos=calculate_point_to_move_towards(p[0.0,0.0,0.0,0.0,0.0,0.0], [0.0,0.0,-1.0], 0.071)
      movel(towardsPos, a=0.15, v=0.1)
      move_thread_flag_4616 = 2
      exit_critical
    end
    move_thread_flag_4616 = 0
    move_thread_han_4616 = run move_thread_4616()
    while (True):
      sleep(1.0E-10)
      if (move_thread_flag_4616 > 1):
        join move_thread_han_4616
        $ 4617 "Until (distance)"
        break
      end
      sync()
    end
    $ 4618 "Direction: Base Z-"
    global move_thread_flag_4618=0
    thread move_thread_4618():
      enter_critical
      move_thread_flag_4618 = 1
      local towardsPos=calculate_point_to_move_towards(p[0.0,0.0,0.0,0.0,0.0,0.0], [0.0,0.0,-1.0], 1000.0)
      movel(towardsPos, a=0.007, v=0.007)
      move_thread_flag_4618 = 2
      exit_critical
    end
    move_thread_flag_4618 = 0
    move_thread_han_4618 = run move_thread_4618()
    while (True):
      local targetTcpDirection=get_target_tcp_speed()
      local stepsToRetract=tool_contact(direction=targetTcpDirection)
      if (stepsToRetract > 0):
        kill move_thread_han_4618
        stopl(0.02)
        local backTrackMovement=get_actual_joint_positions_history(stepsToRetract)
        local contactPose=get_forward_kin(backTrackMovement)
        local posDir=[targetTcpDirection[0],targetTcpDirection[1],targetTcpDirection[2]]
        local retractTo=contactPose
        if (norm(posDir) > 1e-6):
          local normalizedPosDir=normalize(posDir)
          local additionalRetraction=p[normalizedPosDir[0] * 0.0, normalizedPosDir[1] * 0.0, normalizedPosDir[2] * 0.0, 0, 0, 0]
          retractTo = pose_sub(contactPose, additionalRetraction)
        end
        movel(retractTo, a=0.02, v=0.1)
        $ 4619 "Until (tool_contact_detection)"
        break
      end
      sync()
    end
    $ 4620 "Direction: Base Z+"
    global move_thread_flag_4620=0
    thread move_thread_4620():
      enter_critical
      move_thread_flag_4620 = 1
      local towardsPos=calculate_point_to_move_towards(p[0.0,0.0,0.0,0.0,0.0,0.0], [0.0,0.0,1.0], 0.08)
      movel(towardsPos, a=0.15, v=0.1)
      move_thread_flag_4620 = 2
      exit_critical
    end
    move_thread_flag_4620 = 0
    move_thread_han_4620 = run move_thread_4620()
    while (True):
      sleep(1.0E-10)
      if (move_thread_flag_4620 > 1):
        join move_thread_han_4620
        $ 4621 "Until (distance)"
        break
      end
      sync()
    end
    $ 4622 "AB"
    $ 4623 "'desbaste_inicial'"
    # 'desbaste_inicial'
    $ 4624 "bajada_broca≔p[0,0,-0.008,0,0,0]"
    global bajada_broca=p[0,0,-0.008,0,0,0]
    $ 4625 "barrenos_menos1≔6"
    global barrenos_menos1=6
    $ 4626 "barreno_actual≔0"
    global barreno_actual=0
    $ 4627 "Loop barreno_actual≤barrenos_menos1"
    while (barreno_actual <= barrenos_menos1):
      $ 4628 "Perforacion"
      $ 4629 "MoveL"
      $ 4630 "If barreno_actual≟3"
      if (barreno_actual == 3):
        $ 4631 "barreno_actual≔barreno_actual+2"
        global barreno_actual=barreno_actual+2
      end
      $ 4632 "internos≔interpolate_pose(Linea27_A, Linea27_B, barreno_actual/barrenos_menos1)"
      global internos= interpolate_pose (Linea27_A_p, Linea27_B_p, barreno_actual/barrenos_menos1)
      $ 4633 "internos" "breakAfter"
      movel(internos, a=0.5, v=0.1)
      $ 4634 "'desbaste_inicial'"
      # 'desbaste_inicial'
      $ 4635 "bajada_broca≔p[0,0,-0.024,0,0,0]"
      global bajada_broca=p[0,0,-0.024,0,0,0]
      $ 4636 "bajada≔p[0,0,0.024,0,0,0]"
      global bajada=p[0,0,0.024,0,0,0]
      $ 4637 "Direction: Base Z-"
      global move_thread_flag_4637=0
      thread move_thread_4637():
        enter_critical
        move_thread_flag_4637 = 1
        local towardsPos=calculate_point_to_move_towards(p[0.0,0.0,0.0,0.0,0.0,0.0], [0.0,0.0,-1.0], 0.071)
        movel(towardsPos, a=0.15, v=0.1)
        move_thread_flag_4637 = 2
        exit_critical
      end
      move_thread_flag_4637 = 0
      move_thread_han_4637 = run move_thread_4637()
      while (True):
        sleep(1.0E-10)
        if (move_thread_flag_4637 > 1):
          join move_thread_han_4637
          $ 4638 "Until (distance)"
          break
        end
        sync()
      end
      $ 4639 "Direction: Base Z-"
      global move_thread_flag_4639=0
      thread move_thread_4639():
        enter_critical
        move_thread_flag_4639 = 1
        local towardsPos=calculate_point_to_move_towards(p[0.0,0.0,0.0,0.0,0.0,0.0], [0.0,0.0,-1.0], 1000.0)
        movel(towardsPos, a=0.007, v=0.007)
        move_thread_flag_4639 = 2
        exit_critical
      end
      move_thread_flag_4639 = 0
      move_thread_han_4639 = run move_thread_4639()
      while (True):
        local targetTcpDirection=get_target_tcp_speed()
        local stepsToRetract=tool_contact(direction=targetTcpDirection)
        if (stepsToRetract > 0):
          kill move_thread_han_4639
          stopl(0.02)
          local backTrackMovement=get_actual_joint_positions_history(stepsToRetract)
          local contactPose=get_forward_kin(backTrackMovement)
          local posDir=[targetTcpDirection[0],targetTcpDirection[1],targetTcpDirection[2]]
          local retractTo=contactPose
          if (norm(posDir) > 1e-6):
            local normalizedPosDir=normalize(posDir)
            local additionalRetraction=p[normalizedPosDir[0] * 0.0, normalizedPosDir[1] * 0.0, normalizedPosDir[2] * 0.0, 0, 0, 0]
            retractTo = pose_sub(contactPose, additionalRetraction)
          end
          movel(retractTo, a=0.02, v=0.1)
          $ 4640 "Until (tool_contact_detection)"
          break
        end
        sync()
      end
      $ 4641 "Popup: punto contacto alanzdo"
      popup("punto contacto alanzdo", "Mensaje", False, False, blocking=True)
      $ 4642 "Direction: Base Z+"
      global move_thread_flag_4642=0
      thread move_thread_4642():
        enter_critical
        move_thread_flag_4642 = 1
        local towardsPos=calculate_point_to_move_towards(p[0.0,0.0,0.0,0.0,0.0,0.0], [0.0,0.0,1.0], 0.007)
        movel(towardsPos, a=0.015, v=0.015)
        move_thread_flag_4642 = 2
        exit_critical
      end
      move_thread_flag_4642 = 0
      move_thread_han_4642 = run move_thread_4642()
      while (True):
        sleep(1.0E-10)
        if (move_thread_flag_4642 > 1):
          join move_thread_han_4642
          $ 4643 "Until (distance)"
          break
        end
        sync()
      end
      $ 4644 "Wait: 0.3"
      sleep(0.3)
      $ 4645 "Set CO[1]=Encender"
      set_configurable_digital_out(1, True)
      $ 4646 "Wait: 0.3"
      sleep(0.3)
      $ 4647 "Loop 1 times"
      Loop_142 = 0
      while (Loop_142 < 1):
        $ 4648 "bajar≔pose_add(get_actual_tcp_pose(), bajada_broca)"
        global bajar= pose_add ( get_actual_tcp_pose (), bajada_broca)
        $ 4649 "bajar" "breakAfter"
        movel(bajar, a=0.004, v=0.004)
        $ 4650 "subir≔pose_sub(get_actual_tcp_pose(), bajada_broca)"
        global subir= pose_sub ( get_actual_tcp_pose (), bajada_broca)
        $ 4651 "Direction: Base Z+"
        global move_thread_flag_4651=0
        thread move_thread_4651():
          enter_critical
          move_thread_flag_4651 = 1
          local towardsPos=calculate_point_to_move_towards(p[0.0,0.0,0.0,0.0,0.0,0.0], [0.0,0.0,1.0], 0.002)
          movel(towardsPos, a=0.015, v=0.015)
          move_thread_flag_4651 = 2
          exit_critical
        end
        move_thread_flag_4651 = 0
        move_thread_han_4651 = run move_thread_4651()
        while (True):
          sleep(1.0E-10)
          if (move_thread_flag_4651 > 1):
            join move_thread_han_4651
            $ 4652 "Until (distance)"
            break
          end
          sync()
        end
        $ 4653 "Set CO[1]=Apagar"
        set_configurable_digital_out(1, False)
        $ 4654 "subir" "breakAfter"
        movel(subir, a=0.015, v=0.015)
        $ 4655 "bajada_broca≔pose_sub(bajada_broca, bajada)"
        global bajada_broca= pose_sub (bajada_broca, bajada)
        Loop_142 = Loop_142 + 1
      end
      $ 4656 "Direction: Base Z+"
      global move_thread_flag_4656=0
      thread move_thread_4656():
        enter_critical
        move_thread_flag_4656 = 1
        local towardsPos=calculate_point_to_move_towards(p[0.0,0.0,0.0,0.0,0.0,0.0], [0.0,0.0,1.0], 0.08)
        movel(towardsPos, a=0.15, v=0.1)
        move_thread_flag_4656 = 2
        exit_critical
      end
      move_thread_flag_4656 = 0
      move_thread_han_4656 = run move_thread_4656()
      while (True):
        sleep(1.0E-10)
        if (move_thread_flag_4656 > 1):
          join move_thread_han_4656
          $ 4657 "Until (distance)"
          break
        end
        sync()
      end
      $ 4658 "Set CO[1]=Apagar"
      set_configurable_digital_out(1, False)
      $ 4659 "barreno_actual≔barreno_actual+1"
      global barreno_actual=barreno_actual+1
    end
    $ 4662 "Popup: Linea27 con chica Terminada!"
    popup("Linea27 con chica Terminada!", "Mensaje", False, False, blocking=True)
    $ 4663 "Linea28"
    $ 4664 "Marcar_puntos"
    $ 4665 "MoveL"
    $ 4666 "Linea28_B" "breakAfter"
    movel(Linea28_B_p, a=0.5, v=0.1)
    $ 4667 "bajada_comprobacion"
    $ 4668 "Direction: Base Z-"
    global move_thread_flag_4668=0
    thread move_thread_4668():
      enter_critical
      move_thread_flag_4668 = 1
      local towardsPos=calculate_point_to_move_towards(p[0.0,0.0,0.0,0.0,0.0,0.0], [0.0,0.0,-1.0], 0.071)
      movel(towardsPos, a=0.15, v=0.1)
      move_thread_flag_4668 = 2
      exit_critical
    end
    move_thread_flag_4668 = 0
    move_thread_han_4668 = run move_thread_4668()
    while (True):
      sleep(1.0E-10)
      if (move_thread_flag_4668 > 1):
        join move_thread_han_4668
        $ 4669 "Until (distance)"
        break
      end
      sync()
    end
    $ 4670 "Direction: Base Z-"
    global move_thread_flag_4670=0
    thread move_thread_4670():
      enter_critical
      move_thread_flag_4670 = 1
      local towardsPos=calculate_point_to_move_towards(p[0.0,0.0,0.0,0.0,0.0,0.0], [0.0,0.0,-1.0], 1000.0)
      movel(towardsPos, a=0.007, v=0.007)
      move_thread_flag_4670 = 2
      exit_critical
    end
    move_thread_flag_4670 = 0
    move_thread_han_4670 = run move_thread_4670()
    while (True):
      local targetTcpDirection=get_target_tcp_speed()
      local stepsToRetract=tool_contact(direction=targetTcpDirection)
      if (stepsToRetract > 0):
        kill move_thread_han_4670
        stopl(0.02)
        local backTrackMovement=get_actual_joint_positions_history(stepsToRetract)
        local contactPose=get_forward_kin(backTrackMovement)
        local posDir=[targetTcpDirection[0],targetTcpDirection[1],targetTcpDirection[2]]
        local retractTo=contactPose
        if (norm(posDir) > 1e-6):
          local normalizedPosDir=normalize(posDir)
          local additionalRetraction=p[normalizedPosDir[0] * 0.0, normalizedPosDir[1] * 0.0, normalizedPosDir[2] * 0.0, 0, 0, 0]
          retractTo = pose_sub(contactPose, additionalRetraction)
        end
        movel(retractTo, a=0.02, v=0.1)
        $ 4671 "Until (tool_contact_detection)"
        break
      end
      sync()
    end
    $ 4672 "Direction: Base Z+"
    global move_thread_flag_4672=0
    thread move_thread_4672():
      enter_critical
      move_thread_flag_4672 = 1
      local towardsPos=calculate_point_to_move_towards(p[0.0,0.0,0.0,0.0,0.0,0.0], [0.0,0.0,1.0], 0.08)
      movel(towardsPos, a=0.15, v=0.1)
      move_thread_flag_4672 = 2
      exit_critical
    end
    move_thread_flag_4672 = 0
    move_thread_han_4672 = run move_thread_4672()
    while (True):
      sleep(1.0E-10)
      if (move_thread_flag_4672 > 1):
        join move_thread_han_4672
        $ 4673 "Until (distance)"
        break
      end
      sync()
    end
    $ 4674 "AB"
    $ 4675 "'desbaste_inicial'"
    # 'desbaste_inicial'
    $ 4676 "bajada_broca≔p[0,0,-0.008,0,0,0]"
    global bajada_broca=p[0,0,-0.008,0,0,0]
    $ 4677 "barrenos_menos1≔0"
    global barrenos_menos1=0
    $ 4678 "barreno_actual≔0"
    global barreno_actual=0
    $ 4679 "Loop barreno_actual≤barrenos_menos1"
    while (barreno_actual <= barrenos_menos1):
      $ 4680 "Perforacion"
      $ 4681 "MoveL"
      $ 4686 "Linea28_B" "breakAfter"
      movel(Linea28_B_p, a=0.5, v=0.1)
      $ 4687 "'desbaste_inicial'"
      # 'desbaste_inicial'
      $ 4688 "bajada_broca≔p[0,0,-0.024,0,0,0]"
      global bajada_broca=p[0,0,-0.024,0,0,0]
      $ 4689 "bajada≔p[0,0,0.024,0,0,0]"
      global bajada=p[0,0,0.024,0,0,0]
      $ 4690 "Direction: Base Z-"
      global move_thread_flag_4690=0
      thread move_thread_4690():
        enter_critical
        move_thread_flag_4690 = 1
        local towardsPos=calculate_point_to_move_towards(p[0.0,0.0,0.0,0.0,0.0,0.0], [0.0,0.0,-1.0], 0.071)
        movel(towardsPos, a=0.15, v=0.1)
        move_thread_flag_4690 = 2
        exit_critical
      end
      move_thread_flag_4690 = 0
      move_thread_han_4690 = run move_thread_4690()
      while (True):
        sleep(1.0E-10)
        if (move_thread_flag_4690 > 1):
          join move_thread_han_4690
          $ 4691 "Until (distance)"
          break
        end
        sync()
      end
      $ 4692 "Direction: Base Z-"
      global move_thread_flag_4692=0
      thread move_thread_4692():
        enter_critical
        move_thread_flag_4692 = 1
        local towardsPos=calculate_point_to_move_towards(p[0.0,0.0,0.0,0.0,0.0,0.0], [0.0,0.0,-1.0], 1000.0)
        movel(towardsPos, a=0.007, v=0.007)
        move_thread_flag_4692 = 2
        exit_critical
      end
      move_thread_flag_4692 = 0
      move_thread_han_4692 = run move_thread_4692()
      while (True):
        local targetTcpDirection=get_target_tcp_speed()
        local stepsToRetract=tool_contact(direction=targetTcpDirection)
        if (stepsToRetract > 0):
          kill move_thread_han_4692
          stopl(0.02)
          local backTrackMovement=get_actual_joint_positions_history(stepsToRetract)
          local contactPose=get_forward_kin(backTrackMovement)
          local posDir=[targetTcpDirection[0],targetTcpDirection[1],targetTcpDirection[2]]
          local retractTo=contactPose
          if (norm(posDir) > 1e-6):
            local normalizedPosDir=normalize(posDir)
            local additionalRetraction=p[normalizedPosDir[0] * 0.0, normalizedPosDir[1] * 0.0, normalizedPosDir[2] * 0.0, 0, 0, 0]
            retractTo = pose_sub(contactPose, additionalRetraction)
          end
          movel(retractTo, a=0.02, v=0.1)
          $ 4693 "Until (tool_contact_detection)"
          break
        end
        sync()
      end
      $ 4694 "Popup: punto contacto alanzdo"
      popup("punto contacto alanzdo", "Mensaje", False, False, blocking=True)
      $ 4695 "Direction: Base Z+"
      global move_thread_flag_4695=0
      thread move_thread_4695():
        enter_critical
        move_thread_flag_4695 = 1
        local towardsPos=calculate_point_to_move_towards(p[0.0,0.0,0.0,0.0,0.0,0.0], [0.0,0.0,1.0], 0.01)
        movel(towardsPos, a=0.015, v=0.015)
        move_thread_flag_4695 = 2
        exit_critical
      end
      move_thread_flag_4695 = 0
      move_thread_han_4695 = run move_thread_4695()
      while (True):
        sleep(1.0E-10)
        if (move_thread_flag_4695 > 1):
          join move_thread_han_4695
          $ 4696 "Until (distance)"
          break
        end
        sync()
      end
      $ 4697 "Wait: 0.3"
      sleep(0.3)
      $ 4698 "Set CO[1]=Encender"
      set_configurable_digital_out(1, True)
      $ 4699 "Wait: 0.3"
      sleep(0.3)
      $ 4700 "Loop 1 times"
      Loop_146 = 0
      while (Loop_146 < 1):
        $ 4701 "bajar≔pose_add(get_actual_tcp_pose(), bajada_broca)"
        global bajar= pose_add ( get_actual_tcp_pose (), bajada_broca)
        $ 4702 "bajar" "breakAfter"
        movel(bajar, a=0.004, v=0.004)
        $ 4703 "subir≔pose_sub(get_actual_tcp_pose(), bajada_broca)"
        global subir= pose_sub ( get_actual_tcp_pose (), bajada_broca)
        $ 4704 "Direction: Base Z+"
        global move_thread_flag_4704=0
        thread move_thread_4704():
          enter_critical
          move_thread_flag_4704 = 1
          local towardsPos=calculate_point_to_move_towards(p[0.0,0.0,0.0,0.0,0.0,0.0], [0.0,0.0,1.0], 0.002)
          movel(towardsPos, a=0.015, v=0.015)
          move_thread_flag_4704 = 2
          exit_critical
        end
        move_thread_flag_4704 = 0
        move_thread_han_4704 = run move_thread_4704()
        while (True):
          sleep(1.0E-10)
          if (move_thread_flag_4704 > 1):
            join move_thread_han_4704
            $ 4705 "Until (distance)"
            break
          end
          sync()
        end
        $ 4706 "Set CO[1]=Apagar"
        set_configurable_digital_out(1, False)
        $ 4707 "subir" "breakAfter"
        movel(subir, a=0.015, v=0.015)
        $ 4708 "bajada_broca≔pose_sub(bajada_broca, bajada)"
        global bajada_broca= pose_sub (bajada_broca, bajada)
        Loop_146 = Loop_146 + 1
      end
      $ 4709 "Direction: Base Z+"
      global move_thread_flag_4709=0
      thread move_thread_4709():
        enter_critical
        move_thread_flag_4709 = 1
        local towardsPos=calculate_point_to_move_towards(p[0.0,0.0,0.0,0.0,0.0,0.0], [0.0,0.0,1.0], 0.08)
        movel(towardsPos, a=0.15, v=0.1)
        move_thread_flag_4709 = 2
        exit_critical
      end
      move_thread_flag_4709 = 0
      move_thread_han_4709 = run move_thread_4709()
      while (True):
        sleep(1.0E-10)
        if (move_thread_flag_4709 > 1):
          join move_thread_han_4709
          $ 4710 "Until (distance)"
          break
        end
        sync()
      end
      $ 4711 "Set CO[1]=Apagar"
      set_configurable_digital_out(1, False)
      $ 4712 "barreno_actual≔barreno_actual+1"
      global barreno_actual=barreno_actual+1
    end
    $ 4715 "Popup: Linea28 con chica Terminada!"
    popup("Linea28 con chica Terminada!", "Mensaje", False, False, blocking=True)
    $ 4780 "Popup: Linea29 con chica Terminada!"
    popup("Linea29 con chica Terminada!", "Mensaje", False, False, blocking=True)
    $ 4845 "Popup: Linea29B con chica Terminada!"
    popup("Linea29B con chica Terminada!", "Mensaje", False, False, blocking=True)
    $ 5333 "'Subprogramas:'"
    # 'Subprogramas:'
  end
end
